// TIA Portal V15 export
// export: Created 2018-05-29T12:25:38.1552518Z, ExportSetting WithDefaults, DisplayName Totally Integrated Automation Portal, DisplayVersion V15, DisplayName STEP 7 Professional, DisplayVersion V15, DisplayName WinCC Professional, DisplayVersion V15, DisplayName TIA Portal Openness, DisplayVersion V15
FUNCTION "test_stl" : Void   // FC1, STL
{ S7_Optimized_Access := 'TRUE' }
VERSION : 0.1
// stored: AutoNumber true, UDAEnableTagReadback false
   VAR_INPUT
      test : Bool;
   END_VAR
BEGIN

NETWORK
TITLE = 
      A     #test;
      AN    #test;
      S     #test;


NETWORK
TITLE = 
      A     #test;
      AN    #test;
      S     #test;

      A     #test;
      AN    #test;
      S     #test;



END_FUNCTION
